// TIA Portal V18 export
DATA_BLOCK "Agitator"   // DB124
{ S7_Optimized_Access := 'TRUE' }
VERSION : 0.1
// stored: AutoNumber true, DBAccessibleFromOPCUA true, IsOnlyStoredInLoadMemory false, IsRetainMemResEnabled false, IsWriteProtectedInAS false, MemoryReserve 100
   VAR
      Control : Struct
         A1 : Struct
            "Show ON Button" : Bool;
            "Show OFF Button" : Bool;
            ON : Bool;
            OFF : Bool;
            "ON timer okay" : Bool;
            "Off timer Okay" : Bool;
            "Off hmi" : Bool;
            selected : Bool;
            Run : Bool;
            "ON hmi" : Bool;
         END_STRUCT;
         A2 : Struct
            ON : Bool;
            OFF : Bool;
            "ON hmi" : Bool;
            "ON timer okay" : Bool;
            "Off timer Okay" : Bool;
            selected : Bool;
            "Off hmi" : Bool;
            Run : Bool;
            "Show ON Button" : Bool;
            "Show OFF Button" : Bool;
         END_STRUCT;
         B1 : Struct
            ON : Bool;
            "ON hmi" : Bool;
            OFF : Bool;
            "ON timer okay" : Bool;
            "Off timer Okay" : Bool;
            selected : Bool;
            "Off hmi" : Bool;
            Run : Bool;
            "Show ON Button" : Bool;
            "Show OFF Button" : Bool;
         END_STRUCT;
      END_STRUCT;
   END_VAR
   VAR RETAIN
      "Time" : Struct
         A1 : Struct
            "ON time" : Int;
            "OFF time" : Int;
         END_STRUCT;
         A2 : Struct
            "ON time" : Int;
            "OFF time" : Int;
         END_STRUCT;
         B1 : Struct
            "ON time" : Int;
            "OFF time" : Int;
         END_STRUCT;
      END_STRUCT;
      selection : Struct
         A1 : Int;
         A2 : Int;
         B1 : Int;
      END_STRUCT;
   END_VAR
   VAR
      "Time control" : Struct
         A1 : Struct
            "ON time" : Time;
            "OFF time" : Time;
         END_STRUCT;
         A2 : Struct
            "ON time" : Time;
            "OFF time" : Time;
         END_STRUCT;
         B1 : Struct
            "ON time" : Time;
            "OFF time" : Time;
         END_STRUCT;
      END_STRUCT;
      "ON HMI" : Bool;
      "Display ON Button" : Bool;
      "Display Off Button" : Bool;
      "Run time PV" : Struct
         A1 : Int;
         A2 : Int;
         B1 : Int;
      END_STRUCT;
      "Idle time PV" : Struct
         A1 : Int;
         A2 : Int;
         B1 : Int;
      END_STRUCT;
      "Run time PVms" : Struct
         A1 : DInt;
         A2 : DInt;
         B1 : DInt;
      END_STRUCT;
      "Idle time PVmS" : Struct
         A1 : DInt;
         A2 : DInt;
         B1 : DInt;
      END_STRUCT;
   END_VAR
BEGIN
END_DATA_BLOCK
